PROGRAM Axe_03_X_Laser	
VAR	XLaser:FB_Axe_Ethercat_V3;		B_Reset_Y1:BOOL;		TP_not_machine_en_service: TP;
	ACompleter_X_decoupe_en_cours: BOOL;
END_VAR

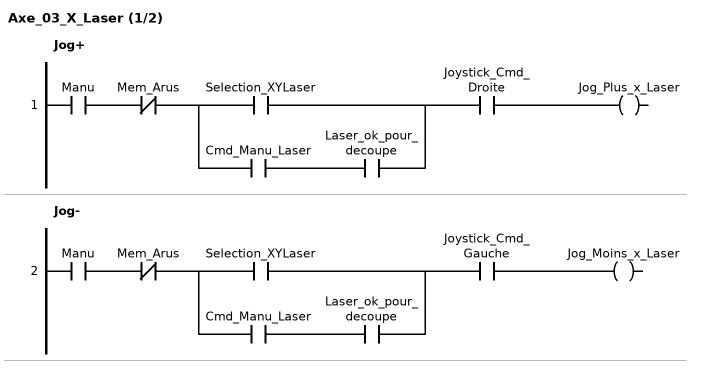
// NETWORK 1: Jog+
Jog_Plus_x_Laser := Manu AND NOT Mem_Arus AND (Selection_XYLaser OR Cmd_Manu_Laser AND Laser_ok_pour_decoupe) AND Joystick_Cmd_Droite;

// NETWORK 2: Jog-
Jog_Moins_x_Laser := Manu AND NOT Mem_Arus AND (Selection_XYLaser OR Cmd_Manu_Laser AND Laser_ok_pour_decoupe) AND Joystick_Cmd_Gauche;

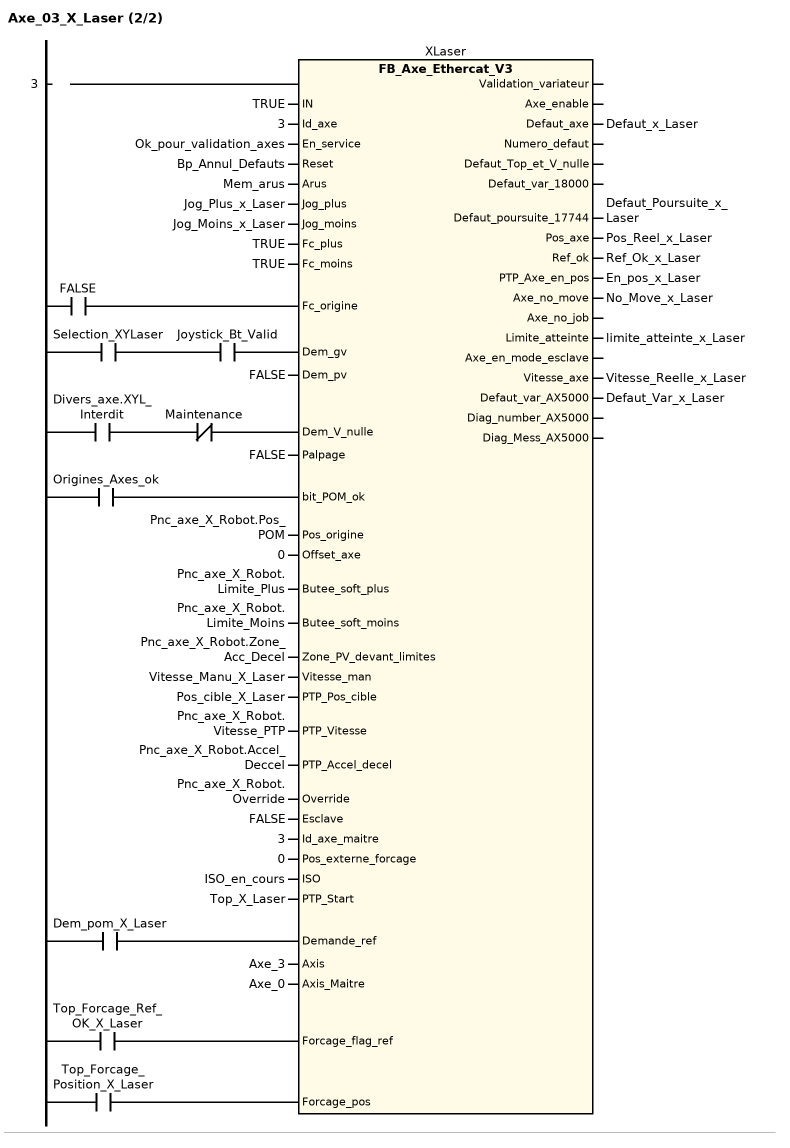
// NETWORK 3
//   Pnc_axe_X_Robot.Pos_POM: 14
//   Pnc_axe_X_Robot.Zone_Acc_Decel: 10
//   Pos_cible_X_Laser: Axe Y Superieur
//   Pnc_axe_X_Robot.Accel_Deccel: 6
//   Pnc_axe_X_Robot.Override: 7
//   Axe_3: ***************************** Variables Axe3---Y1 *****************************
//   Axe_0: Axe bidon mais nécessaire car il est obligatoire de lier un axe maître en entrée de chaque FB_axe
XLaser(
    IN := TRUE,
    Id_axe := 3,
    En_service := Ok_pour_validation_axes,
    Reset := Bp_Annul_Defauts,
    Arus := Mem_arus,
    Jog_plus := Jog_Plus_x_Laser,
    Jog_moins := Jog_Moins_x_Laser,
    Fc_plus := TRUE,
    Fc_moins := TRUE,
    Fc_origine := FALSE,
    Dem_gv := Selection_XYLaser AND Joystick_Bt_Valid,
    Dem_pv := FALSE,
    Dem_V_nulle := Divers_axe.XYL_Interdit AND NOT Maintenance,
    Palpage := FALSE,
    bit_POM_ok := Origines_Axes_ok,
    Pos_origine := Pnc_axe_X_Robot.Pos_POM,
    Offset_axe := 0,
    Butee_soft_plus := Pnc_axe_X_Robot.Limite_Plus,
    Butee_soft_moins := Pnc_axe_X_Robot.Limite_Moins,
    Zone_PV_devant_limites := Pnc_axe_X_Robot.Zone_Acc_Decel,
    Vitesse_man := Vitesse_Manu_X_Laser,
    PTP_Pos_cible := Pos_cible_X_Laser,
    PTP_Vitesse := Pnc_axe_X_Robot.Vitesse_PTP,
    PTP_Accel_decel := Pnc_axe_X_Robot.Accel_Deccel,
    Override := Pnc_axe_X_Robot.Override,
    Esclave := FALSE,
    Id_axe_maitre := 3,
    Pos_externe_forcage := 0,
    ISO := ISO_en_cours,
    PTP_Start := Top_X_Laser,
    Demande_ref := Dem_pom_X_Laser,
    Axis := Axe_3,
    Axis_Maitre := Axe_0,
    Forcage_flag_ref := Top_Forcage_Ref_OK_X_Laser,
    Forcage_pos := Top_Forcage_Position_X_Laser,
    Defaut_axe => Defaut_x_Laser,
    Defaut_poursuite_17744 => Defaut_Poursuite_x_Laser,
    Pos_axe => Pos_Reel_x_Laser,
    Ref_ok => Ref_Ok_x_Laser,
    PTP_Axe_en_pos => En_pos_x_Laser,
    Axe_no_move => No_Move_x_Laser,
    Limite_atteinte => limite_atteinte_x_Laser,
    Vitesse_axe => Vitesse_Reelle_x_Laser,
    Defaut_var_AX5000 => Defaut_Var_x_Laser); // FB_Axe_Ethercat_V3

END_PROGRAM

(* stored: Version 1.1.0.1
   POU Axe_03_X_Laser: Id {9c0050db-ead0-409e-89a1-77ba75ec6eca}, SpecialFunc None *)
